PROGRAM Dock_State
VAR
END_VAR

IF Shuttle.LoadDistance[1] < 30000 THEN
	
	Shuttle.IsDocked[1]		:= TRUE;
	Shuttle.IsNotDocked[1] 	:= FALSE;
	
ELSE
	
	Shuttle.IsDocked[1]		:= FALSE;
	Shuttle.IsNotDocked[1] 	:= TRUE;

END_IF

IF Shuttle.LoadDistance[2] < 30000 THEN
	
	Shuttle.IsDocked[2]		:= TRUE;
	Shuttle.IsNotDocked[2] 	:= FALSE;
	
ELSE
	
	Shuttle.IsDocked[2]		:= FALSE;
	Shuttle.IsNotDocked[2] 	:= TRUE;

END_IF

IF Shuttle.IsDocked[1] AND Shuttle.IsDocked[2] THEN
	
	Shuttle.IsCompletelyDocked		:= TRUE;
	Shuttle.IsNotCompletelyDocked	:= FALSE;

ELSE 
	
	Shuttle.IsCompletelyDocked		:= FALSE;
	Shuttle.IsNotCompletelyDocked	:= TRUE;

END_IF

END_PROGRAM

(* stored: Version 1.1.0.1, ProductVersion 3.1.4024.9
   POU Dock_State: Id {c2f9a6a6-1478-4500-9ce0-2bb70b8e8847}, SpecialFunc None *)
